LIN {X 0,Y 142.327,Z 764.935,A -85,B 0,C 180,E1 7207.887,E2 7207.887} C_VEL
LIN {X 0,Y 140.279,Z 766.739,A -85,B 0,C 180,E1 7204.976,E2 7204.976} C_VEL
LIN {X 0,Y 137.442,Z 769.448,A -85,B 0,C 180,E1 7201.685,E2 7201.685} C_VEL
LIN {X 0,Y 130.762,Z 776.335,A -85,B 0,C 180,E1 7194.167,E2 7194.167} C_VEL
LIN {X 0,Y 129.959,Z 778.072,A -85,B 0,C 180,E1 7191.372,E2 7191.372} C_VEL
LIN {X 0,Y 136.056,Z 784.68,A -85,B 0,C 180,E1 7176.161,E2 7176.161} C_VEL
LIN {X 0,Y 149.948,Z 789.28,A -85,B 0,C 180,E1 7165.01,E2 7165.01} C_VEL
LIN {X 0,Y 152.41,Z 789.916,A -85,B 0,C 180,E1 7163.584,E2 7163.584} C_VEL
LIN {X 0,Y 141.835,Z 799.917,A -85,B 0,C 180,E1 7157.151,E2 7157.151} C_VEL
LIN {X 0,Y 132.635,Z 808.523,A -85,B 0,C 180,E1 7149.289,E2 7149.289} C_VEL
LIN {X 0,Y 125.571,Z 815.712,A -85,B 0,C 180,E1 7139.786,E2 7139.786} C_VEL
LIN {X 0,Y 121.824,Z 820.643,A -85,B 0,C 180,E1 7130.164,E2 7130.164} C_VEL
LIN {X 0,Y 120.73,Z 823.658,A -85,B 0,C 180,E1 7120.981,E2 7120.981} C_VEL
LIN {X 0,Y 120.991,Z 824.935,A -85,B 0,C 180,E1 7113.791,E2 7113.791} C_VEL
LIN {X 0,Y 121.063,Z 825.276,A -85,B 0,C 180,E1 7108.107,E2 7108.107} C_VEL
LIN {X 0,Y 120.709,Z 824.803,A -85,B 0,C 180,E1 7101.425,E2 7101.425} C_VEL
LIN {X 0,Y 121.285,Z 822.901,A -85,B 0,C 180,E1 7092.24,E2 7092.24} C_VEL
LIN {X 0,Y 124.517,Z 819.128,A -85,B 0,C 180,E1 7082.242,E2 7082.242} C_VEL
LIN {X 0,Y 130.8,Z 813.597,A -85,B 0,C 180,E1 7072.85,E2 7072.85} C_VEL
LIN {X 0,Y 139.988,Z 806.145,A -85,B 0,C 180,E1 7064.418,E2 7064.418} C_VEL
LIN {X 0,Y 151.07,Z 797.105,A -85,B 0,C 180,E1 7057.417,E2 7057.417} C_VEL
LIN {X 0,Y 163.41,Z 786.509,A -85,B 0,C 180,E1 7051.635,E2 7051.635} C_VEL
LIN {X 0,Y 148.498,Z 786.74,A -85,B 0,C 180,E1 7044.634,E2 7044.634} C_VEL
LIN {X 0,Y 138.257,Z 785.962,A -85,B 0,C 180,E1 7036.381,E2 7036.381} C_VEL
LIN {X 0,Y 132.254,Z 784.513,A -85,B 0,C 180,E1 7026.51,E2 7026.51} C_VEL
LIN {X 0,Y 131.134,Z 783.114,A -85,B 0,C 180,E1 7018.688,E2 7018.688} C_VEL
LIN {X 0,Y 134.316,Z 780.824,A -85,B 0,C 180,E1 7007.531,E2 7007.531} C_VEL
LIN {X 0,Y 143.154,Z 778.008,A -85,B 0,C 180,E1 6997.408,E2 6997.408} C_VEL
LIN {X 0,Y 155.053,Z 775.028,A -85,B 0,C 180,E1 6989.801,E2 6989.801} C_VEL
LIN {X 0,Y 165.287,Z 772.555,A -85,B 0,C 180,E1 6985.356,E2 6985.356} C_VEL
LIN {X 0,Y 153.328,Z 781.917,A -85,B 0,C 180,E1 6979.727,E2 6979.727} C_VEL
LIN {X 0,Y 142.444,Z 789.724,A -85,B 0,C 180,E1 6972.913,E2 6972.913} C_VEL
LIN {X 0,Y 133.258,Z 795.917,A -85,B 0,C 180,E1 6964.768,E2 6964.768} C_VEL
LIN {X 0,Y 126.676,Z 800.222,A -85,B 0,C 180,E1 6955.73,E2 6955.73} C_VEL
LIN {X 0,Y 122.964,Z 802.645,A -85,B 0,C 180,E1 6946.535,E2 6946.535} C_VEL
LIN {X 0,Y 121.464,Z 803.514,A -85,B 0,C 180,E1 6937.569,E2 6937.569} C_VEL
LIN {X 0,Y 121.376,Z 803.12,A -85,B 0,C 180,E1 6929.056,E2 6929.056} C_VEL
LIN {X 0,Y 122.613,Z 801.434,A -85,B 0,C 180,E1 6920.14,E2 6920.14} C_VEL
LIN {X 0,Y 125.928,Z 798.163,A -85,B 0,C 180,E1 6911.002,E2 6911.002} C_VEL
LIN {X 0,Y 131.607,Z 793.272,A -85,B 0,C 180,E1 6902.391,E2 6902.391} C_VEL
LIN {X 0,Y 140.034,Z 786.271,A -85,B 0,C 180,E1 6894.162,E2 6894.162} C_VEL
LIN {X 0,Y 149.617,Z 778.131,A -85,B 0,C 180,E1 6887.549,E2 6887.549} C_VEL
LIN {X 0,Y 160.16,Z 768.649,A -85,B 0,C 180,E1 6882.02,E2 6882.02} C_VEL
LIN {X 0,Y 171.365,Z 757.748,A -85,B 0,C 180,E1 6877.361,E2 6877.361} C_VEL
LIN {X 0,Y 183.117,Z 745.114,A -85,B 0,C 180,E1 6873.301,E2 6873.301} C_VEL
LIN {X 0,Y 172.911,Z 750.159,A -85,B 0,C 180,E1 6870.589,E2 6870.589} C_VEL
LIN {X 0,Y 159.994,Z 756.362,A -85,B 0,C 180,E1 6865.854,E2 6865.854} C_VEL
LIN {X 0,Y 149.86,Z 761.284,A -85,B 0,C 180,E1 6860.71,E2 6860.71} C_VEL
LIN {X 0,Y 142.024,Z 765.507,A -85,B 0,C 180,E1 6855.1,E2 6855.1} C_VEL
LIN {X 0,Y 136.055,Z 769.276,A -85,B 0,C 180,E1 6848.879,E2 6848.879} C_VEL
LIN {X 0,Y 132.224,Z 772.647,A -85,B 0,C 180,E1 6842.602,E2 6842.602} C_VEL
LIN {X 0,Y 130.123,Z 776.685,A -85,B 0,C 180,E1 6834.269,E2 6834.269} C_VEL
LIN {X 0,Y 129.959,Z 778.072,A -85,B 0,C 180,E1 6831.372,E2 6831.372} C_VEL
LIN {X 0,Y 129.127,Z 780.467,A -85,B 0,C 180,E1 6827.59,E2 6827.59} C_VEL
LIN {X 0,Y 127.185,Z 786.25,A -85,B 0,C 180,E1 6819.802,E2 6819.802} C_VEL
LIN {X 0,Y 128.371,Z 787.985,A -85,B 0,C 180,E1 6816.472,E2 6816.472} C_VEL
LIN {X 0,Y 128.538,Z 788.078,A -85,B 0,C 180,E1 6816.241,E2 6816.241} C_VEL
LIN {X 0,Y 141.942,Z 792.523,A -85,B 0,C 180,E1 6804.718,E2 6804.718} C_VEL
LIN {X 0,Y 143.15,Z 792.902,A -85,B 0,C 180,E1 6803.903,E2 6803.903} C_VEL
LIN {X 0,Y 131.986,Z 802.686,A -85,B 0,C 180,E1 6796.657,E2 6796.657} C_VEL
LIN {X 0,Y 122.988,Z 810.577,A -85,B 0,C 180,E1 6788.16,E2 6788.16} C_VEL
LIN {X 0,Y 116.513,Z 816.869,A -85,B 0,C 180,E1 6778.163,E2 6778.163} C_VEL
LIN {X 0,Y 113.291,Z 821.249,A -85,B 0,C 180,E1 6767.611,E2 6767.611} C_VEL
LIN {X 0,Y 112.786,Z 823.617,A -85,B 0,C 180,E1 6758.154,E2 6758.154} C_VEL
LIN {X 0,Y 113.119,Z 824.457,A -85,B 0,C 180,E1 6751.519,E2 6751.519} C_VEL
LIN {X 0,Y 112.949,Z 824.477,A -85,B 0,C 180,E1 6745.43,E2 6745.43} C_VEL
LIN {X 0,Y 112.786,Z 823.47,A -85,B 0,C 180,E1 6736.674,E2 6736.674} C_VEL
LIN {X 0,Y 114.786,Z 820.705,A -85,B 0,C 180,E1 6726.147,E2 6726.147} C_VEL
LIN {X 0,Y 120.346,Z 815.871,A -85,B 0,C 180,E1 6715.334,E2 6715.334} C_VEL
LIN {X 0,Y 129.16,Z 809.22,A -85,B 0,C 180,E1 6705.835,E2 6705.835} C_VEL
LIN {X 0,Y 140.544,Z 800.671,A -85,B 0,C 180,E1 6697.844,E2 6697.844} C_VEL
LIN {X 0,Y 153.385,Z 790.579,A -85,B 0,C 180,E1 6691.431,E2 6691.431} C_VEL
LIN {X 0,Y 139.962,Z 790.459,A -85,B 0,C 180,E1 6684.476,E2 6684.476} C_VEL
LIN {X 0,Y 130.135,Z 789.445,A -85,B 0,C 180,E1 6675.598,E2 6675.598} C_VEL
LIN {X 0,Y 125.2,Z 788.207,A -85,B 0,C 180,E1 6666.878,E2 6666.878} C_VEL
LIN {X 0,Y 124.752,Z 785.827,A -85,B 0,C 180,E1 6653.093,E2 6653.093} C_VEL
LIN {X 0,Y 134.755,Z 782.281,A -85,B 0,C 180,E1 6637.763,E2 6637.763} C_VEL
LIN {X 0,Y 148.914,Z 778.871,A -85,B 0,C 180,E1 6628.416,E2 6628.416} C_VEL
LIN {X 0,Y 155.328,Z 777.427,A -85,B 0,C 180,E1 6625.483,E2 6625.483} C_VEL
LIN {X 0,Y 142.741,Z 786.385,A -85,B 0,C 180,E1 6619.158,E2 6619.158} C_VEL
LIN {X 0,Y 132.024,Z 793.328,A -85,B 0,C 180,E1 6611.794,E2 6611.794} C_VEL
LIN {X 0,Y 123.207,Z 798.686,A -85,B 0,C 180,E1 6602.938,E2 6602.938} C_VEL
LIN {X 0,Y 117.214,Z 802.205,A -85,B 0,C 180,E1 6593.104,E2 6593.104} C_VEL
LIN {X 0,Y 114.199,Z 803.931,A -85,B 0,C 180,E1 6583.159,E2 6583.159} C_VEL
LIN {X 0,Y 113.323,Z 804.205,A -85,B 0,C 180,E1 6574.048,E2 6574.048} C_VEL
LIN {X 0,Y 113.769,Z 803.328,A -85,B 0,C 180,E1 6564.958,E2 6564.958} C_VEL
LIN {X 0,Y 115.926,Z 801.107,A -85,B 0,C 180,E1 6555.515,E2 6555.515} C_VEL
LIN {X 0,Y 120.867,Z 796.979,A -85,B 0,C 180,E1 6545.567,E2 6545.567} C_VEL
LIN {X 0,Y 128.146,Z 791.351,A -85,B 0,C 180,E1 6536.895,E2 6536.895} C_VEL
LIN {X 0,Y 137.71,Z 783.926,A -85,B 0,C 180,E1 6529.197,E2 6529.197} C_VEL
LIN {X 0,Y 148.674,Z 774.977,A -85,B 0,C 180,E1 6522.787,E2 6522.787} C_VEL
LIN {X 0,Y 160.252,Z 764.773,A -85,B 0,C 180,E1 6517.59,E2 6517.59} C_VEL
LIN {X 0,Y 172.115,Z 753.272,A -85,B 0,C 180,E1 6513.296,E2 6513.296} C_VEL
LIN {X 0,Y 156.016,Z 760.477,A -85,B 0,C 180,E1 6507.895,E2 6507.895} C_VEL
LIN {X 0,Y 144.573,Z 765.541,A -85,B 0,C 180,E1 6502.359,E2 6502.359} C_VEL
LIN {X 0,Y 136.263,Z 769.637,A -85,B 0,C 180,E1 6496.63,E2 6496.63} C_VEL
LIN {X 0,Y 129.858,Z 773.325,A -85,B 0,C 180,E1 6490.202,E2 6490.202} C_VEL
LIN {X 0,Y 125.481,Z 776.754,A -85,B 0,C 180,E1 6483.199,E2 6483.199} C_VEL
LIN {X 0,Y 123.17,Z 780.474,A -85,B 0,C 180,E1 6474.879,E2 6474.879} C_VEL
LIN {X 0,Y 124.08,Z 784.569,A -85,B 0,C 180,E1 6465.059,E2 6465.059} C_VEL
LIN {X 0,Y 128.538,Z 788.078,A -85,B 0,C 180,E1 6456.241,E2 6456.241} C_VEL
LIN {X 0,Y 129.404,Z 789.371,A -85,B 0,C 180,E1 6454.005,E2 6454.005} C_VEL
LIN {X 0,Y 129.566,Z 793.797,A -85,B 0,C 180,E1 6448.256,E2 6448.256} C_VEL
LIN {X 0,Y 131.281,Z 794.906,A -85,B 0,C 180,E1 6446.152,E2 6446.152} C_VEL
LIN {X 0,Y 133.864,Z 795.665,A -85,B 0,C 180,E1 6444.259,E2 6444.259} C_VEL
LIN {X 0,Y 122.64,Z 804.754,A -85,B 0,C 180,E1 6436.519,E2 6436.519} C_VEL
LIN {X 0,Y 113.746,Z 812.064,A -85,B 0,C 180,E1 6427.339,E2 6427.339} C_VEL
LIN {X 0,Y 107.834,Z 817.537,A -85,B 0,C 180,E1 6417.022,E2 6417.022} C_VEL
LIN {X 0,Y 105.071,Z 821.303,A -85,B 0,C 180,E1 6406.019,E2 6406.019} C_VEL
LIN {X 0,Y 104.914,Z 823.292,A -85,B 0,C 180,E1 6396.017,E2 6396.017} C_VEL
LIN {X 0,Y 105.176,Z 823.802,A -85,B 0,C 180,E1 6389.455,E2 6389.455} C_VEL
LIN {X 0,Y 104.791,Z 823.598,A -85,B 0,C 180,E1 6382.323,E2 6382.323} C_VEL
LIN {X 0,Y 105.338,Z 821.994,A -85,B 0,C 180,E1 6371.745,E2 6371.745} C_VEL
LIN {X 0,Y 109.014,Z 818.561,A -85,B 0,C 180,E1 6360.311,E2 6360.311} C_VEL
LIN {X 0,Y 116.195,Z 813.317,A -85,B 0,C 180,E1 6349.805,E2 6349.805} C_VEL
LIN {X 0,Y 126.551,Z 806.237,A -85,B 0,C 180,E1 6340.669,E2 6340.669} C_VEL
LIN {X 0,Y 138.833,Z 797.607,A -85,B 0,C 180,E1 6333.339,E2 6333.339} C_VEL
LIN {X 0,Y 143.313,Z 794.292,A -85,B 0,C 180,E1 6331.198,E2 6331.198} C_VEL
LIN {X 0,Y 129.824,Z 793.788,A -85,B 0,C 180,E1 6323.126,E2 6323.126} C_VEL
LIN {X 0,Y 118.498,Z 791.93,A -85,B 0,C 180,E1 6308.734,E2 6308.734} C_VEL
LIN {X 0,Y 117.735,Z 789.183,A -85,B 0,C 180,E1 6292.189,E2 6292.189} C_VEL
LIN {X 0,Y 128.54,Z 785.675,A -85,B 0,C 180,E1 6276.139,E2 6276.139} C_VEL
LIN {X 0,Y 144.073,Z 782.191,A -85,B 0,C 180,E1 6266.274,E2 6266.274} C_VEL
LIN {X 0,Y 145.349,Z 781.942,A -85,B 0,C 180,E1 6265.638,E2 6265.638} C_VEL
LIN {X 0,Y 132.716,Z 790.085,A -85,B 0,C 180,E1 6258.885,E2 6258.885} C_VEL
LIN {X 0,Y 121.618,Z 796.572,A -85,B 0,C 180,E1 6250.503,E2 6250.503} C_VEL
LIN {X 0,Y 113.234,Z 801.123,A -85,B 0,C 180,E1 6240.807,E2 6240.807} C_VEL
LIN {X 0,Y 107.93,Z 803.88,A -85,B 0,C 180,E1 6230.046,E2 6230.046} C_VEL
LIN {X 0,Y 105.668,Z 804.929,A -85,B 0,C 180,E1 6219.257,E2 6219.257} C_VEL
LIN {X 0,Y 105.392,Z 804.699,A -85,B 0,C 180,E1 6210,E2 6210} C_VEL
LIN {X 0,Y 106.563,Z 803.319,A -85,B 0,C 180,E1 6200.277,E2 6200.277} C_VEL
LIN {X 0,Y 110.166,Z 800.347,A -85,B 0,C 180,E1 6189.825,E2 6189.825} C_VEL
LIN {X 0,Y 116.875,Z 795.483,A -85,B 0,C 180,E1 6179.686,E2 6179.686} C_VEL
LIN {X 0,Y 125.861,Z 789.097,A -85,B 0,C 180,E1 6171.128,E2 6171.128} C_VEL
LIN {X 0,Y 136.419,Z 781.311,A -85,B 0,C 180,E1 6164.088,E2 6164.088} C_VEL
LIN {X 0,Y 148.581,Z 771.642,A -85,B 0,C 180,E1 6158.062,E2 6158.062} C_VEL
LIN {X 0,Y 161.347,Z 760.482,A -85,B 0,C 180,E1 6153.142,E2 6153.142} C_VEL
LIN {X 0,Y 151.263,Z 764.693,A -85,B 0,C 180,E1 6149.721,E2 6149.721} C_VEL
LIN {X 0,Y 139.888,Z 769.384,A -85,B 0,C 180,E1 6144.493,E2 6144.493} C_VEL
LIN {X 0,Y 130.482,Z 773.549,A -85,B 0,C 180,E1 6138.313,E2 6138.313} C_VEL
LIN {X 0,Y 123.628,Z 777.186,A -85,B 0,C 180,E1 6131.667,E2 6131.667} C_VEL
LIN {X 0,Y 118.817,Z 780.496,A -85,B 0,C 180,E1 6124.345,E2 6124.345} C_VEL
LIN {X 0,Y 116.124,Z 784.251,A -85,B 0,C 180,E1 6115.062,E2 6115.062} C_VEL
LIN {X 0,Y 117.022,Z 788.236,A -85,B 0,C 180,E1 6104.643,E2 6104.643} C_VEL
LIN {X 0,Y 124.71,Z 792.903,A -85,B 0,C 180,E1 6091.771,E2 6091.771} C_VEL
LIN {X 0,Y 131.281,Z 794.906,A -85,B 0,C 180,E1 6086.152,E2 6086.152} C_VEL
LIN {X 0,Y 131.585,Z 795.64,A -85,B 0,C 180,E1 6085.153,E2 6085.153} C_VEL
LIN {X 0,Y 130.245,Z 797.057,A -85,B 0,C 180,E1 6083.974,E2 6083.974} C_VEL
LIN {X 0,Y 126.747,Z 799.167,A -85,B 0,C 180,E1 6082.605,E2 6082.605} C_VEL
LIN {X 0,Y 118.25,Z 803.234,A -85,B 0,C 180,E1 6080.011,E2 6080.011} C_VEL
LIN {X 0,Y 116.114,Z 804.555,A -85,B 0,C 180,E1 6078.768,E2 6078.768} C_VEL
LIN {X 0,Y 106.417,Z 811.832,A -85,B 0,C 180,E1 6069.014,E2 6069.014} C_VEL
LIN {X 0,Y 99.818,Z 817.385,A -85,B 0,C 180,E1 6057.437,E2 6057.437} C_VEL
LIN {X 0,Y 97.024,Z 820.956,A -85,B 0,C 180,E1 6045.541,E2 6045.541} C_VEL
LIN {X 0,Y 96.982,Z 822.68,A -85,B 0,C 180,E1 6035.324,E2 6035.324} C_VEL
LIN {X 0,Y 97.205,Z 823.082,A -85,B 0,C 180,E1 6029.41,E2 6029.41} C_VEL
LIN {X 0,Y 96.815,Z 822.91,A -85,B 0,C 180,E1 6022.284,E2 6022.284} C_VEL
LIN {X 0,Y 97.474,Z 821.379,A -85,B 0,C 180,E1 6010.837,E2 6010.837} C_VEL
LIN {X 0,Y 101.605,Z 818.045,A -85,B 0,C 180,E1 5998.563,E2 5998.563} C_VEL
LIN {X 0,Y 109.495,Z 812.893,A -85,B 0,C 180,E1 5987.488,E2 5987.488} C_VEL
LIN {X 0,Y 120.665,Z 805.879,A -85,B 0,C 180,E1 5978.075,E2 5978.075} C_VEL
LIN {X 0,Y 133.116,Z 797.639,A -85,B 0,C 180,E1 5970.855,E2 5970.855} C_VEL
LIN {X 0,Y 119.37,Z 796.719,A -85,B 0,C 180,E1 5961.109,E2 5961.109} C_VEL
LIN {X 0,Y 110.948,Z 795.031,A -85,B 0,C 180,E1 5948.289,E2 5948.289} C_VEL
LIN {X 0,Y 110.474,Z 792.426,A -85,B 0,C 180,E1 5931.672,E2 5931.672} C_VEL
LIN {X 0,Y 121.869,Z 788.946,A -85,B 0,C 180,E1 5914.744,E2 5914.744} C_VEL
LIN {X 0,Y 135.348,Z 786.121,A -85,B 0,C 180,E1 5905.832,E2 5905.832} C_VEL
LIN {X 0,Y 122.667,Z 793.471,A -85,B 0,C 180,E1 5898.582,E2 5898.582} C_VEL
LIN {X 0,Y 111.691,Z 799.236,A -85,B 0,C 180,E1 5889.465,E2 5889.465} C_VEL
LIN {X 0,Y 103.665,Z 803.11,A -85,B 0,C 180,E1 5878.833,E2 5878.833} C_VEL
LIN {X 0,Y 99.147,Z 805.155,A -85,B 0,C 180,E1 5867.611,E2 5867.611} C_VEL
LIN {X 0,Y 97.511,Z 805.715,A -85,B 0,C 180,E1 5857.068,E2 5857.068} C_VEL
LIN {X 0,Y 97.599,Z 805.136,A -85,B 0,C 180,E1 5847.064,E2 5847.064} C_VEL
LIN {X 0,Y 99.603,Z 803.296,A -85,B 0,C 180,E1 5836.059,E2 5836.059} C_VEL
LIN {X 0,Y 104.469,Z 799.877,A -85,B 0,C 180,E1 5825.095,E2 5825.095} C_VEL
LIN {X 0,Y 112.23,Z 794.841,A -85,B 0,C 180,E1 5815.237,E2 5815.237} C_VEL
LIN {X 0,Y 122.526,Z 788.079,A -85,B 0,C 180,E1 5806.727,E2 5806.727} C_VEL
LIN {X 0,Y 134.885,Z 779.433,A -85,B 0,C 180,E1 5799.563,E2 5799.563} C_VEL
LIN {X 0,Y 148.116,Z 769.16,A -85,B 0,C 180,E1 5793.868,E2 5793.868} C_VEL
LIN {X 0,Y 150.282,Z 767.348,A -85,B 0,C 180,E1 5793.065,E2 5793.065} C_VEL
LIN {X 0,Y 134.711,Z 773.297,A -85,B 0,C 180,E1 5786.447,E2 5786.447} C_VEL
LIN {X 0,Y 124.392,Z 777.425,A -85,B 0,C 180,E1 5779.873,E2 5779.873} C_VEL
LIN {X 0,Y 117.351,Z 780.792,A -85,B 0,C 180,E1 5773.302,E2 5773.302} C_VEL
LIN {X 0,Y 111.904,Z 784.218,A -85,B 0,C 180,E1 5765.128,E2 5765.128} C_VEL
LIN {X 0,Y 108.991,Z 787.657,A -85,B 0,C 180,E1 5755.793,E2 5755.793} C_VEL
LIN {X 0,Y 109.85,Z 791.651,A -85,B 0,C 180,E1 5744.155,E2 5744.155} C_VEL
LIN {X 0,Y 117.483,Z 796.065,A -85,B 0,C 180,E1 5730.983,E2 5730.983} C_VEL
LIN {X 0,Y 124.676,Z 798.141,A -85,B 0,C 180,E1 5724.733,E2 5724.733} C_VEL
LIN {X 0,Y 116.114,Z 804.555,A -85,B 0,C 180,E1 5718.768,E2 5718.768} C_VEL
LIN {X 0,Y 111.632,Z 807.293,A -85,B 0,C 180,E1 5715.891,E2 5715.891} C_VEL
LIN {X 0,Y 97.65,Z 813.239,A -85,B 0,C 180,E1 5707.704,E2 5707.704} C_VEL
LIN {X 0,Y 94.735,Z 814.833,A -85,B 0,C 180,E1 5704.259,E2 5704.259} C_VEL
LIN {X 0,Y 89.936,Z 819.134,A -85,B 0,C 180,E1 5691.523,E2 5691.523} C_VEL
LIN {X 0,Y 88.829,Z 821.577,A -85,B 0,C 180,E1 5679.066,E2 5679.066} C_VEL
LIN {X 0,Y 89.213,Z 822.314,A -85,B 0,C 180,E1 5671.284,E2 5671.284} C_VEL
LIN {X 0,Y 88.99,Z 822.354,A -85,B 0,C 180,E1 5664.843,E2 5664.843} C_VEL
LIN {X 0,Y 89.061,Z 821.415,A -85,B 0,C 180,E1 5653.7,E2 5653.7} C_VEL
LIN {X 0,Y 92.282,Z 818.805,A -85,B 0,C 180,E1 5640.819,E2 5640.819} C_VEL
LIN {X 0,Y 99.688,Z 814.332,A -85,B 0,C 180,E1 5628.549,E2 5628.549} C_VEL
LIN {X 0,Y 111.313,Z 807.695,A -85,B 0,C 180,E1 5617.771,E2 5617.771} C_VEL
LIN {X 0,Y 123.104,Z 800.647,A -85,B 0,C 180,E1 5610.526,E2 5610.526} C_VEL
LIN {X 0,Y 110.365,Z 799.48,A -85,B 0,C 180,E1 5600.135,E2 5600.135} C_VEL
LIN {X 0,Y 103.467,Z 797.974,A -85,B 0,C 180,E1 5588.333,E2 5588.333} C_VEL
LIN {X 0,Y 103.134,Z 795.448,A -85,B 0,C 180,E1 5571.074,E2 5571.074} C_VEL
LIN {X 0,Y 115.694,Z 791.888,A -85,B 0,C 180,E1 5552.737,E2 5552.737} C_VEL
LIN {X 0,Y 125.218,Z 790.042,A -85,B 0,C 180,E1 5546.015,E2 5546.015} C_VEL
LIN {X 0,Y 112.006,Z 796.859,A -85,B 0,C 180,E1 5537.811,E2 5537.811} C_VEL
LIN {X 0,Y 101.314,Z 801.806,A -85,B 0,C 180,E1 5527.726,E2 5527.726} C_VEL
LIN {X 0,Y 93.907,Z 804.94,A -85,B 0,C 180,E1 5515.884,E2 5515.884} C_VEL
LIN {X 0,Y 90.253,Z 806.307,A -85,B 0,C 180,E1 5503.453,E2 5503.453} C_VEL
LIN {X 0,Y 89.401,Z 806.281,A -85,B 0,C 180,E1 5492.564,E2 5492.564} C_VEL
LIN {X 0,Y 90.262,Z 805.262,A -85,B 0,C 180,E1 5481.721,E2 5481.721} C_VEL
LIN {X 0,Y 93.906,Z 802.719,A -85,B 0,C 180,E1 5469.429,E2 5469.429} C_VEL
LIN {X 0,Y 101.16,Z 798.371,A -85,B 0,C 180,E1 5457.742,E2 5457.742} C_VEL
LIN {X 0,Y 111.001,Z 792.525,A -85,B 0,C 180,E1 5448.197,E2 5448.197} C_VEL
LIN {X 0,Y 123.162,Z 784.885,A -85,B 0,C 180,E1 5440.26,E2 5440.26} C_VEL
LIN {X 0,Y 136.367,Z 775.768,A -85,B 0,C 180,E1 5434.052,E2 5434.052} C_VEL
LIN {X 0,Y 139.253,Z 773.525,A -85,B 0,C 180,E1 5432.806,E2 5432.806} C_VEL
LIN {X 0,Y 128.944,Z 777.191,A -85,B 0,C 180,E1 5428.232,E2 5428.232} C_VEL
LIN {X 0,Y 119.028,Z 780.834,A -85,B 0,C 180,E1 5422.212,E2 5422.212} C_VEL
LIN {X 0,Y 110.702,Z 784.375,A -85,B 0,C 180,E1 5414.651,E2 5414.651} C_VEL
LIN {X 0,Y 105.118,Z 787.545,A -85,B 0,C 180,E1 5406.556,E2 5406.556} C_VEL
LIN {X 0,Y 101.745,Z 791.023,A -85,B 0,C 180,E1 5396.058,E2 5396.058} C_VEL
LIN {X 0,Y 102.408,Z 794.702,A -85,B 0,C 180,E1 5384.137,E2 5384.137} C_VEL
LIN {X 0,Y 111.081,Z 799.293,A -85,B 0,C 180,E1 5369.134,E2 5369.134} C_VEL
LIN {X 0,Y 115.287,Z 800.561,A -85,B 0,C 180,E1 5365.158,E2 5365.158} C_VEL
LIN {X 0,Y 103.854,Z 808.358,A -85,B 0,C 180,E1 5356.12,E2 5356.12} C_VEL
LIN {X 0,Y 94.957,Z 814.662,A -85,B 0,C 180,E1 5344.653,E2 5344.653} C_VEL
LIN {X 0,Y 94.735,Z 814.833,A -85,B 0,C 180,E1 5344.259,E2 5344.259} C_VEL
LIN {X 0,Y 91.625,Z 816.539,A -85,B 0,C 180,E1 5340.012,E2 5340.012} C_VEL
LIN {X 0,Y 84.273,Z 818.948,A -85,B 0,C 180,E1 5331.523,E2 5331.523} C_VEL
LIN {X 0,Y 81.129,Z 820.124,A -85,B 0,C 180,E1 5324.927,E2 5324.927} C_VEL
LIN {X 0,Y 80.882,Z 820.397,A -85,B 0,C 180,E1 5322.967,E2 5322.967} C_VEL
LIN {X 0,Y 81.168,Z 821.517,A -85,B 0,C 180,E1 5312.824,E2 5312.824} C_VEL
LIN {X 0,Y 81.157,Z 821.671,A -85,B 0,C 180,E1 5307.175,E2 5307.175} C_VEL
LIN {X 0,Y 80.91,Z 821.063,A -85,B 0,C 180,E1 5295.69,E2 5295.69} C_VEL
LIN {X 0,Y 83.789,Z 818.853,A -85,B 0,C 180,E1 5281.489,E2 5281.489} C_VEL
LIN {X 0,Y 91.227,Z 814.826,A -85,B 0,C 180,E1 5268.043,E2 5268.043} C_VEL
LIN {X 0,Y 102.576,Z 809.014,A -85,B 0,C 180,E1 5256.937,E2 5256.937} C_VEL
LIN {X 0,Y 112.986,Z 803.32,A -85,B 0,C 180,E1 5250.053,E2 5250.053} C_VEL
LIN {X 0,Y 98.12,Z 801.427,A -85,B 0,C 180,E1 5234.154,E2 5234.154} C_VEL
LIN {X 0,Y 94.598,Z 799.248,A -85,B 0,C 180,E1 5217.575,E2 5217.575} C_VEL
LIN {X 0,Y 100.27,Z 796.673,A -85,B 0,C 180,E1 5200.786,E2 5200.786} C_VEL
LIN {X 0,Y 115.285,Z 793.547,A -85,B 0,C 180,E1 5186.368,E2 5186.368} C_VEL
LIN {X 0,Y 101.905,Z 799.653,A -85,B 0,C 180,E1 5177.382,E2 5177.382} C_VEL
LIN {X 0,Y 91.4,Z 803.887,A -85,B 0,C 180,E1 5166.209,E2 5166.209} C_VEL
LIN {X 0,Y 84.56,Z 806.349,A -85,B 0,C 180,E1 5152.968,E2 5152.968} C_VEL
LIN {X 0,Y 81.781,Z 807.116,A -85,B 0,C 180,E1 5139.856,E2 5139.856} C_VEL
LIN {X 0,Y 81.588,Z 806.709,A -85,B 0,C 180,E1 5127.893,E2 5127.893} C_VEL
LIN {X 0,Y 83.604,Z 805.194,A -85,B 0,C 180,E1 5115.455,E2 5115.455} C_VEL
LIN {X 0,Y 89.096,Z 802.065,A -85,B 0,C 180,E1 5102.606,E2 5102.606} C_VEL
LIN {X 0,Y 97.926,Z 797.337,A -85,B 0,C 180,E1 5091.477,E2 5091.477} C_VEL
LIN {X 0,Y 110.125,Z 790.535,A -85,B 0,C 180,E1 5081.883,E2 5081.883} C_VEL
LIN {X 0,Y 123.847,Z 782.156,A -85,B 0,C 180,E1 5074.565,E2 5074.565} C_VEL
LIN {X 0,Y 128.184,Z 779.257,A -85,B 0,C 180,E1 5072.637,E2 5072.637} C_VEL
LIN {X 0,Y 113.405,Z 784.188,A -85,B 0,C 180,E1 5064.483,E2 5064.483} C_VEL
LIN {X 0,Y 104.295,Z 787.633,A -85,B 0,C 180,E1 5056.526,E2 5056.526} C_VEL
LIN {X 0,Y 98.041,Z 790.777,A -85,B 0,C 180,E1 5047.621,E2 5047.621} C_VEL
LIN {X 0,Y 94.456,Z 794.024,A -85,B 0,C 180,E1 5036.968,E2 5036.968} C_VEL
LIN {X 0,Y 95.069,Z 797.698,A -85,B 0,C 180,E1 5023.505,E2 5023.505} C_VEL
LIN {X 0,Y 103.869,Z 802.001,A -85,B 0,C 180,E1 5007.898,E2 5007.898} C_VEL
LIN {X 0,Y 105.931,Z 802.689,A -85,B 0,C 180,E1 5005.68,E2 5005.68} C_VEL
LIN {X 0,Y 94.058,Z 810.122,A -85,B 0,C 180,E1 4995.448,E2 4995.448} C_VEL
LIN {X 0,Y 85.508,Z 815.736,A -85,B 0,C 180,E1 4982.662,E2 4982.662} C_VEL
LIN {X 0,Y 81.378,Z 819.418,A -85,B 0,C 180,E1 4968.63,E2 4968.63} C_VEL
LIN {X 0,Y 80.882,Z 820.397,A -85,B 0,C 180,E1 4962.967,E2 4962.967} C_VEL
LIN {X 0,Y 79.979,Z 820.962,A -85,B 0,C 180,E1 4958.291,E2 4958.291} C_VEL
LIN {X 0,Y 77.39,Z 821.241,A -85,B 0,C 180,E1 4952.047,E2 4952.047} C_VEL
LIN {X 0,Y 72.904,Z 820.718,A -85,B 0,C 180,E1 4938.383,E2 4938.383} C_VEL
LIN {X 0,Y 72.882,Z 820.566,A -85,B 0,C 180,E1 4936.572,E2 4936.572} C_VEL
LIN {X 0,Y 75.796,Z 818.577,A -85,B 0,C 180,E1 4920.785,E2 4920.785} C_VEL
LIN {X 0,Y 83.72,Z 814.783,A -85,B 0,C 180,E1 4906.156,E2 4906.156} C_VEL
LIN {X 0,Y 96.448,Z 808.907,A -85,B 0,C 180,E1 4893.968,E2 4893.968} C_VEL
LIN {X 0,Y 102.951,Z 805.671,A -85,B 0,C 180,E1 4889.528,E2 4889.528} C_VEL
LIN {X 0,Y 89.162,Z 803.541,A -85,B 0,C 180,E1 4871.643,E2 4871.643} C_VEL
LIN {X 0,Y 88.461,Z 800.706,A -85,B 0,C 180,E1 4848.919,E2 4848.919} C_VEL
LIN {X 0,Y 103.066,Z 797.216,A -85,B 0,C 180,E1 4828.406,E2 4828.406} C_VEL
LIN {X 0,Y 105.229,Z 796.833,A -85,B 0,C 180,E1 4826.738,E2 4826.738} C_VEL
LIN {X 0,Y 91.78,Z 802.191,A -85,B 0,C 180,E1 4816.879,E2 4816.879} C_VEL
LIN {X 0,Y 81.508,Z 805.728,A -85,B 0,C 180,E1 4804.353,E2 4804.353} C_VEL
LIN {X 0,Y 75.369,Z 807.536,A -85,B 0,C 180,E1 4789.37,E2 4789.37} C_VEL
LIN {X 0,Y 73.511,Z 807.79,A -85,B 0,C 180,E1 4775.464,E2 4775.464} C_VEL
LIN {X 0,Y 74.167,Z 807.024,A -85,B 0,C 180,E1 4762.253,E2 4762.253} C_VEL
LIN {X 0,Y 78.21,Z 804.759,A -85,B 0,C 180,E1 4747.448,E2 4747.448} C_VEL
LIN {X 0,Y 86.547,Z 800.711,A -85,B 0,C 180,E1 4733.9,E2 4733.9} C_VEL
LIN {X 0,Y 98.37,Z 794.853,A -85,B 0,C 180,E1 4722.96,E2 4722.96} C_VEL
LIN {X 0,Y 112.017,Z 787.456,A -85,B 0,C 180,E1 4714.796,E2 4714.796} C_VEL
LIN {X 0,Y 117.162,Z 784.41,A -85,B 0,C 180,E1 4712.305,E2 4712.305} C_VEL
LIN {X 0,Y 100.165,Z 789.885,A -85,B 0,C 180,E1 4701.063,E2 4701.063} C_VEL
LIN {X 0,Y 87.1,Z 796.784,A -85,B 0,C 180,E1 4678.029,E2 4678.029} C_VEL
LIN {X 0,Y 87.663,Z 800.478,A -85,B 0,C 180,E1 4662.752,E2 4662.752} C_VEL
LIN {X 0,Y 96.693,Z 804.518,A -85,B 0,C 180,E1 4646.414,E2 4646.414} C_VEL
LIN {X 0,Y 84.657,Z 811.405,A -85,B 0,C 180,E1 4635.124,E2 4635.124} C_VEL
LIN {X 0,Y 76.638,Z 816.282,A -85,B 0,C 180,E1 4621.457,E2 4621.457} C_VEL
LIN {X 0,Y 73.066,Z 819.447,A -85,B 0,C 180,E1 4605.884,E2 4605.884} C_VEL
LIN {X 0,Y 73.139,Z 820.743,A -85,B 0,C 180,E1 4593.706,E2 4593.706} C_VEL
LIN {X 0,Y 73.208,Z 820.941,A -85,B 0,C 180,E1 4587.651,E2 4587.651} C_VEL
LIN {X 0,Y 72.882,Z 820.566,A -85,B 0,C 180,E1 4576.572,E2 4576.572} C_VEL
LIN {X 0,Y 72.451,Z 819.941,A -85,B 0,C 180,E1 4570.485,E2 4570.485} C_VEL
LIN {X 0,Y 70.778,Z 817.93,A -85,B 0,C 180,E1 4557.608,E2 4557.608} C_VEL
LIN {X 0,Y 72.248,Z 816.416,A -85,B 0,C 180,E1 4550.168,E2 4550.168} C_VEL
LIN {X 0,Y 73.097,Z 816.013,A -85,B 0,C 180,E1 4548.567,E2 4548.567} C_VEL
LIN {X 0,Y 85.17,Z 811.104,A -85,B 0,C 180,E1 4534.736,E2 4534.736} C_VEL
LIN {X 0,Y 93.005,Z 807.723,A -85,B 0,C 180,E1 4528.93,E2 4528.93} C_VEL
LIN {X 0,Y 81.228,Z 805.699,A -85,B 0,C 180,E1 4511.356,E2 4511.356} C_VEL
LIN {X 0,Y 80.942,Z 802.997,A -85,B 0,C 180,E1 4487.875,E2 4487.875} C_VEL
LIN {X 0,Y 95.146,Z 799.794,A -85,B 0,C 180,E1 4467.215,E2 4467.215} C_VEL
LIN {X 0,Y 81.624,Z 804.484,A -85,B 0,C 180,E1 4456.281,E2 4456.281} C_VEL
LIN {X 0,Y 71.664,Z 807.341,A -85,B 0,C 180,E1 4442.018,E2 4442.018} C_VEL
LIN {X 0,Y 66.546,Z 808.499,A -85,B 0,C 180,E1 4425.692,E2 4425.692} C_VEL
LIN {X 0,Y 65.517,Z 808.383,A -85,B 0,C 180,E1 4410.875,E2 4410.875} C_VEL
LIN {X 0,Y 67.204,Z 807.216,A -85,B 0,C 180,E1 4396.229,E2 4396.229} C_VEL
LIN {X 0,Y 73.127,Z 804.534,A -85,B 0,C 180,E1 4380.513,E2 4380.513} C_VEL
LIN {X 0,Y 83.595,Z 800.051,A -85,B 0,C 180,E1 4367.018,E2 4367.018} C_VEL
LIN {X 0,Y 97.275,Z 793.703,A -85,B 0,C 180,E1 4356.703,E2 4356.703} C_VEL
LIN {X 0,Y 105.982,Z 789.198,A -85,B 0,C 180,E1 4351.997,E2 4351.997} C_VEL
LIN {X 0,Y 91.639,Z 793.536,A -85,B 0,C 180,E1 4341.106,E2 4341.106} C_VEL
LIN {X 0,Y 84.052,Z 796.452,A -85,B 0,C 180,E1 4330.975,E2 4330.975} C_VEL
LIN {X 0,Y 79.591,Z 799.445,A -85,B 0,C 180,E1 4318.563,E2 4318.563} C_VEL
LIN {X 0,Y 80.204,Z 803.047,A -85,B 0,C 180,E1 4301.843,E2 4301.843} C_VEL
LIN {X 0,Y 87.254,Z 806.3,A -85,B 0,C 180,E1 4287.105,E2 4287.105} C_VEL
LIN {X 0,Y 75.265,Z 812.451,A -85,B 0,C 180,E1 4274.755,E2 4274.755} C_VEL
LIN {X 0,Y 67.538,Z 816.799,A -85,B 0,C 180,E1 4259.144,E2 4259.144} C_VEL
LIN {X 0,Y 64.904,Z 819.328,A -85,B 0,C 180,E1 4242.455,E2 4242.455} C_VEL
LIN {X 0,Y 65.307,Z 820.172,A -85,B 0,C 180,E1 4230.877,E2 4230.877} C_VEL
LIN {X 0,Y 64.94,Z 820.193,A -85,B 0,C 180,E1 4222.924,E2 4222.924} C_VEL
LIN {X 0,Y 66.011,Z 819.153,A -85,B 0,C 180,E1 4206.807,E2 4206.807} C_VEL
LIN {X 0,Y 72.483,Z 816.272,A -85,B 0,C 180,E1 4189.583,E2 4189.583} C_VEL
LIN {X 0,Y 73.097,Z 816.013,A -85,B 0,C 180,E1 4188.567,E2 4188.567} C_VEL
LIN {X 0,Y 74.535,Z 815.053,A -85,B 0,C 180,E1 4184.736,E2 4184.736} C_VEL
LIN {X 0,Y 76.604,Z 812.162,A -85,B 0,C 180,E1 4174.079,E2 4174.079} C_VEL
LIN {X 0,Y 78.834,Z 811.083,A -85,B 0,C 180,E1 4171.31,E2 4171.31} C_VEL
LIN {X 0,Y 82.983,Z 809.464,A -85,B 0,C 180,E1 4168.026,E2 4168.026} C_VEL
LIN {X 0,Y 73.452,Z 807.708,A -85,B 0,C 180,E1 4151.779,E2 4151.779} C_VEL
LIN {X 0,Y 73.658,Z 804.965,A -85,B 0,C 180,E1 4125.854,E2 4125.854} C_VEL
LIN {X 0,Y 84.877,Z 802.539,A -85,B 0,C 180,E1 4107.709,E2 4107.709} C_VEL
LIN {X 0,Y 71.433,Z 806.475,A -85,B 0,C 180,E1 4095.55,E2 4095.55} C_VEL
LIN {X 0,Y 61.897,Z 808.721,A -85,B 0,C 180,E1 4078.987,E2 4078.987} C_VEL
LIN {X 0,Y 57.908,Z 809.3,A -85,B 0,C 180,E1 4060.949,E2 4060.949} C_VEL
LIN {X 0,Y 57.856,Z 808.786,A -85,B 0,C 180,E1 4045.043,E2 4045.043} C_VEL
LIN {X 0,Y 61.631,Z 807.069,A -85,B 0,C 180,E1 4027.085,E2 4027.085} C_VEL
LIN {X 0,Y 70.796,Z 803.595,A -85,B 0,C 180,E1 4010.54,E2 4010.54} C_VEL
LIN {X 0,Y 83.497,Z 798.556,A -85,B 0,C 180,E1 3998.516,E2 3998.516} C_VEL
LIN {X 0,Y 94.845,Z 793.489,A -85,B 0,C 180,E1 3991.445,E2 3991.445} C_VEL
LIN {X 0,Y 78.01,Z 798.608,A -85,B 0,C 180,E1 3974.856,E2 3974.856} C_VEL
LIN {X 0,Y 71.9,Z 804.825,A -85,B 0,C 180,E1 3943.855,E2 3943.855} C_VEL
LIN {X 0,Y 78.006,Z 807.799,A -85,B 0,C 180,E1 3928.156,E2 3928.156} C_VEL
LIN {X 0,Y 65.861,Z 813.343,A -85,B 0,C 180,E1 3914.294,E2 3914.294} C_VEL
LIN {X 0,Y 58.361,Z 817.25,A -85,B 0,C 180,E1 3895.36,E2 3895.36} C_VEL
LIN {X 0,Y 56.983,Z 819.125,A -85,B 0,C 180,E1 3877.055,E2 3877.055} C_VEL
LIN {X 0,Y 57.322,Z 819.481,A -85,B 0,C 180,E1 3869,E2 3869} C_VEL
LIN {X 0,Y 57.01,Z 819.206,A -85,B 0,C 180,E1 3854.697,E2 3854.697} C_VEL
LIN {X 0,Y 61.162,Z 817.404,A -85,B 0,C 180,E1 3835.098,E2 3835.098} C_VEL
LIN {X 0,Y 71.405,Z 813.794,A -85,B 0,C 180,E1 3818.357,E2 3818.357} C_VEL
LIN {X 0,Y 78.834,Z 811.083,A -85,B 0,C 180,E1 3811.31,E2 3811.31} C_VEL
LIN {X 0,Y 79.417,Z 810.557,A -85,B 0,C 180,E1 3809.717,E2 3809.717} C_VEL
LIN {X 0,Y 78.414,Z 810.141,A -85,B 0,C 180,E1 3807.5,E2 3807.5} C_VEL
LIN {X 0,Y 75.387,Z 809.933,A -85,B 0,C 180,E1 3804.493,E2 3804.493} C_VEL
LIN {X 0,Y 67.936,Z 809.967,A -85,B 0,C 180,E1 3797.862,E2 3797.862} C_VEL
LIN {X 0,Y 66.426,Z 809.758,A -85,B 0,C 180,E1 3795.024,E2 3795.024} C_VEL
LIN {X 0,Y 66.126,Z 806.799,A -85,B 0,C 180,E1 3764.203,E2 3764.203} C_VEL
LIN {X 0,Y 74.93,Z 804.917,A -85,B 0,C 180,E1 3748.637,E2 3748.637} C_VEL
LIN {X 0,Y 60.656,Z 808.337,A -85,B 0,C 180,E1 3733.816,E2 3733.816} C_VEL
LIN {X 0,Y 52.25,Z 809.816,A -85,B 0,C 180,E1 3714.898,E2 3714.898} C_VEL
LIN {X 0,Y 49.603,Z 809.909,A -85,B 0,C 180,E1 3695.785,E2 3695.785} C_VEL
LIN {X 0,Y 50.757,Z 809.148,A -85,B 0,C 180,E1 3677.486,E2 3677.486} C_VEL
LIN {X 0,Y 56.828,Z 807.052,A -85,B 0,C 180,E1 3658.141,E2 3658.141} C_VEL
LIN {X 0,Y 68.628,Z 803.091,A -85,B 0,C 180,E1 3642.01,E2 3642.01} C_VEL
LIN {X 0,Y 83.651,Z 797.417,A -85,B 0,C 180,E1 3630.962,E2 3630.962} C_VEL
LIN {X 0,Y 64.839,Z 803.717,A -85,B 0,C 180,E1 3602.655,E2 3602.655} C_VEL
LIN {X 0,Y 65.151,Z 807.442,A -85,B 0,C 180,E1 3579.334,E2 3579.334} C_VEL
LIN {X 0,Y 68.75,Z 809.13,A -85,B 0,C 180,E1 3569.466,E2 3569.466} C_VEL
LIN {X 0,Y 55.951,Z 814.265,A -85,B 0,C 180,E1 3552.771,E2 3552.771} C_VEL
LIN {X 0,Y 49.574,Z 817.384,A -85,B 0,C 180,E1 3531.287,E2 3531.287} C_VEL
LIN {X 0,Y 49.268,Z 818.704,A -85,B 0,C 180,E1 3512.326,E2 3512.326} C_VEL
LIN {X 0,Y 49.132,Z 818.771,A -85,B 0,C 180,E1 3505.634,E2 3505.634} C_VEL
LIN {X 0,Y 50.08,Z 818.09,A -85,B 0,C 180,E1 3485.211,E2 3485.211} C_VEL
LIN {X 0,Y 57.985,Z 815.649,A -85,B 0,C 180,E1 3463.595,E2 3463.595} C_VEL
LIN {X 0,Y 71.544,Z 811.454,A -85,B 0,C 180,E1 3448.302,E2 3448.302} C_VEL
LIN {X 0,Y 72.985,Z 810.964,A -85,B 0,C 180,E1 3447.021,E2 3447.021} C_VEL
LIN {X 0,Y 66.426,Z 809.758,A -85,B 0,C 180,E1 3435.024,E2 3435.024} C_VEL
LIN {X 0,Y 63.703,Z 809.344,A -85,B 0,C 180,E1 3428.613,E2 3428.613} C_VEL
LIN {X 0,Y 57.455,Z 808.961,A -85,B 0,C 180,E1 3409.842,E2 3409.842} C_VEL
LIN {X 0,Y 58.378,Z 808.47,A -85,B 0,C 180,E1 3402.799,E2 3402.799} C_VEL
LIN {X 0,Y 64.664,Z 807.13,A -85,B 0,C 180,E1 3389.591,E2 3389.591} C_VEL
LIN {X 0,Y 50.413,Z 809.811,A -85,B 0,C 180,E1 3372.403,E2 3372.403} C_VEL
LIN {X 0,Y 42.833,Z 810.696,A -85,B 0,C 180,E1 3349.076,E2 3349.076} C_VEL
LIN {X 0,Y 41.723,Z 810.413,A -85,B 0,C 180,E1 3327.253,E2 3327.253} C_VEL
LIN {X 0,Y 45.713,Z 809.078,A -85,B 0,C 180,E1 3304.059,E2 3304.059} C_VEL
LIN {X 0,Y 56.671,Z 805.965,A -85,B 0,C 180,E1 3283.666,E2 3283.666} C_VEL
LIN {X 0,Y 71.128,Z 801.393,A -85,B 0,C 180,E1 3270.965,E2 3270.965} C_VEL
LIN {X 0,Y 72.453,Z 800.923,A -85,B 0,C 180,E1 3270.02,E2 3270.02} C_VEL
LIN {X 0,Y 57.041,Z 805.886,A -85,B 0,C 180,E1 3243.018,E2 3243.018} C_VEL
LIN {X 0,Y 57.328,Z 809.161,A -85,B 0,C 180,E1 3218.518,E2 3218.518} C_VEL
LIN {X 0,Y 59.523,Z 810.208,A -85,B 0,C 180,E1 3211.184,E2 3211.184} C_VEL
LIN {X 0,Y 47.002,Z 814.607,A -85,B 0,C 180,E1 3192.901,E2 3192.901} C_VEL
LIN {X 0,Y 41.137,Z 817.283,A -85,B 0,C 180,E1 3166.957,E2 3166.957} C_VEL
LIN {X 0,Y 41.402,Z 818.028,A -85,B 0,C 180,E1 3149.999,E2 3149.999} C_VEL
LIN {X 0,Y 41.338,Z 817.789,A -85,B 0,C 180,E1 3130.206,E2 3130.206} C_VEL
LIN {X 0,Y 48.004,Z 816.063,A -85,B 0,C 180,E1 3104.912,E2 3104.912} C_VEL
LIN {X 0,Y 61.684,Z 812.555,A -85,B 0,C 180,E1 3086.933,E2 3086.933} C_VEL
LIN {X 0,Y 62.968,Z 812.17,A -85,B 0,C 180,E1 3085.685,E2 3085.685} C_VEL
LIN {X 0,Y 56.055,Z 809.576,A -85,B 0,C 180,E1 3055.518,E2 3055.518} C_VEL
LIN {X 0,Y 58.378,Z 808.47,A -85,B 0,C 180,E1 3042.799,E2 3042.799} C_VEL
LIN {X 0,Y 58.581,Z 808.346,A -85,B 0,C 180,E1 3039.409,E2 3039.409} C_VEL
LIN {X 0,Y 57.12,Z 808.573,A -85,B 0,C 180,E1 3035.093,E2 3035.093} C_VEL
LIN {X 0,Y 53.821,Z 809.18,A -85,B 0,C 180,E1 3029.859,E2 3029.859} C_VEL
LIN {X 0,Y 47.493,Z 810.182,A -85,B 0,C 180,E1 3022.123,E2 3022.123} C_VEL
LIN {X 0,Y 38.736,Z 811.189,A -85,B 0,C 180,E1 3006.637,E2 3006.637} C_VEL
LIN {X 0,Y 33.834,Z 811.376,A -85,B 0,C 180,E1 2980.214,E2 2980.214} C_VEL
LIN {X 0,Y 34.858,Z 810.763,A -85,B 0,C 180,E1 2955.04,E2 2955.04} C_VEL
LIN {X 0,Y 43.468,Z 808.715,A -85,B 0,C 180,E1 2928.16,E2 2928.16} C_VEL
LIN {X 0,Y 58.68,Z 804.813,A -85,B 0,C 180,E1 2910.747,E2 2910.747} C_VEL
LIN {X 0,Y 61.056,Z 804.109,A -85,B 0,C 180,E1 2908.893,E2 2908.893} C_VEL
LIN {X 0,Y 48.836,Z 810.352,A -85,B 0,C 180,E1 2860.355,E2 2860.355} C_VEL
LIN {X 0,Y 50.418,Z 811.107,A -85,B 0,C 180,E1 2853.599,E2 2853.599} C_VEL
LIN {X 0,Y 37.097,Z 815.082,A -85,B 0,C 180,E1 2830.306,E2 2830.306} C_VEL
LIN {X 0,Y 32.983,Z 816.973,A -85,B 0,C 180,E1 2800.479,E2 2800.479} C_VEL
LIN {X 0,Y 33.303,Z 817.31,A -85,B 0,C 180,E1 2788.279,E2 2788.279} C_VEL
LIN {X 0,Y 34.791,Z 816.869,A -85,B 0,C 180,E1 2758.848,E2 2758.848} C_VEL
LIN {X 0,Y 45.911,Z 814.66,A -85,B 0,C 180,E1 2731.857,E2 2731.857} C_VEL
LIN {X 0,Y 53.065,Z 813.073,A -85,B 0,C 180,E1 2723.775,E2 2723.775} C_VEL
LIN {X 0,Y 50.462,Z 809.952,A -85,B 0,C 180,E1 2681.513,E2 2681.513} C_VEL
LIN {X 0,Y 54.563,Z 809.058,A -85,B 0,C 180,E1 2671.139,E2 2671.139} C_VEL
LIN {X 0,Y 40.672,Z 811.016,A -85,B 0,C 180,E1 2651.588,E2 2651.588} C_VEL
LIN {X 0,Y 38.736,Z 811.189,A -85,B 0,C 180,E1 2646.637,E2 2646.637} C_VEL
LIN {X 0,Y 35.1,Z 811.509,A -85,B 0,C 180,E1 2636.967,E2 2636.967} C_VEL
LIN {X 0,Y 29.535,Z 811.819,A -85,B 0,C 180,E1 2619.62,E2 2619.62} C_VEL
LIN {X 0,Y 27.272,Z 811.543,A -85,B 0,C 180,E1 2592.274,E2 2592.274} C_VEL
LIN {X 0,Y 28.364,Z 811.253,A -85,B 0,C 180,E1 2584.454,E2 2584.454} C_VEL
LIN {X 0,Y 40.058,Z 809.021,A -85,B 0,C 180,E1 2556.991,E2 2556.991} C_VEL
LIN {X 0,Y 49.768,Z 806.879,A -85,B 0,C 180,E1 2546.88,E2 2546.88} C_VEL
LIN {X 0,Y 41.071,Z 811.725,A -85,B 0,C 180,E1 2498.587,E2 2498.587} C_VEL
LIN {X 0,Y 41.293,Z 811.878,A -85,B 0,C 180,E1 2496.943,E2 2496.943} C_VEL
LIN {X 0,Y 28.094,Z 815.103,A -85,B 0,C 180,E1 2469.837,E2 2469.837} C_VEL
LIN {X 0,Y 25.234,Z 816.55,A -85,B 0,C 180,E1 2432.27,E2 2432.27} C_VEL
LIN {X 0,Y 25.058,Z 816.583,A -85,B 0,C 180,E1 2423.124,E2 2423.124} C_VEL
LIN {X 0,Y 30.109,Z 815.824,A -85,B 0,C 180,E1 2383.063,E2 2383.063} C_VEL
LIN {X 0,Y 43.31,Z 813.691,A -85,B 0,C 180,E1 2360.795,E2 2360.795} C_VEL
LIN {X 0,Y 43.832,Z 810.854,A -85,B 0,C 180,E1 2315.752,E2 2315.752} C_VEL
LIN {X 0,Y 44.643,Z 810.689,A -85,B 0,C 180,E1 2313.623,E2 2313.623} C_VEL
LIN {X 0,Y 30.36,Z 812.083,A -85,B 0,C 180,E1 2288.737,E2 2288.737} C_VEL
LIN {X 0,Y 25.698,Z 812.03,A -85,B 0,C 180,E1 2256.704,E2 2256.704} C_VEL
LIN {X 0,Y 28.364,Z 811.253,A -85,B 0,C 180,E1 2224.454,E2 2224.454} C_VEL
LIN {X 0,Y 29.828,Z 810.911,A -85,B 0,C 180,E1 2214.61,E2 2214.61} C_VEL
LIN {X 0,Y 34.824,Z 809.971,A -85,B 0,C 180,E1 2188.866,E2 2188.866} C_VEL
LIN {X 0,Y 37.63,Z 809.446,A -85,B 0,C 180,E1 2184.982,E2 2184.982} C_VEL
LIN {X 0,Y 38.346,Z 809.318,A -85,B 0,C 180,E1 2184.011,E2 2184.011} C_VEL
LIN {X 0,Y 32.281,Z 812.483,A -85,B 0,C 180,E1 2142.103,E2 2142.103} C_VEL
LIN {X 0,Y 18.636,Z 815.119,A -85,B 0,C 180,E1 2106.168,E2 2106.168} C_VEL
LIN {X 0,Y 17.301,Z 815.851,A -85,B 0,C 180,E1 2069.999,E2 2069.999} C_VEL
LIN {X 0,Y 21.766,Z 815.463,A -85,B 0,C 180,E1 2018.653,E2 2018.653} C_VEL
LIN {X 0,Y 33.626,Z 814.062,A -85,B 0,C 180,E1 1996.095,E2 1996.095} C_VEL
LIN {X 0,Y 34.511,Z 812.118,A -85,B 0,C 180,E1 1957.265,E2 1957.265} C_VEL
LIN {X 0,Y 20.517,Z 812.868,A -85,B 0,C 180,E1 1925.791,E2 1925.791} C_VEL
LIN {X 0,Y 18.037,Z 812.544,A -85,B 0,C 180,E1 1880.428,E2 1880.428} C_VEL
LIN {X 0,Y 27.074,Z 811.204,A -85,B 0,C 180,E1 1839.147,E2 1839.147} C_VEL
LIN {X 0,Y 37.63,Z 809.446,A -85,B 0,C 180,E1 1824.982,E2 1824.982} C_VEL
LIN {X 0,Y 38.325,Z 809.347,A -85,B 0,C 180,E1 1822.476,E2 1822.476} C_VEL
LIN {X 0,Y 37.662,Z 809.561,A -85,B 0,C 180,E1 1818.513,E2 1818.513} C_VEL
LIN {X 0,Y 35.206,Z 810.201,A -85,B 0,C 180,E1 1812.495,E2 1812.495} C_VEL
LIN {X 0,Y 29.832,Z 811.543,A -85,B 0,C 180,E1 1802.713,E2 1802.713} C_VEL
LIN {X 0,Y 25.284,Z 812.519,A -85,B 0,C 180,E1 1794.22,E2 1794.22} C_VEL
LIN {X 0,Y 21.88,Z 813.138,A -85,B 0,C 180,E1 1789.001,E2 1789.001} C_VEL
LIN {X 0,Y 9.143,Z 814.957,A -85,B 0,C 180,E1 1729.149,E2 1729.149} C_VEL
LIN {X 0,Y 9.213,Z 815.12,A -85,B 0,C 180,E1 1709.997,E2 1709.997} C_VEL
LIN {X 0,Y 19.101,Z 814.653,A -85,B 0,C 180,E1 1635.162,E2 1635.162} C_VEL
LIN {X 0,Y 24.352,Z 814.171,A -85,B 0,C 180,E1 1627.681,E2 1627.681} C_VEL
LIN {X 0,Y 24.913,Z 813.296,A -85,B 0,C 180,E1 1604.414,E2 1604.414} C_VEL
LIN {X 0,Y 11.068,Z 813.544,A -85,B 0,C 180,E1 1562.825,E2 1562.825} C_VEL
LIN {X 0,Y 12.646,Z 813.003,A -85,B 0,C 180,E1 1490.765,E2 1490.765} C_VEL
LIN {X 0,Y 27.35,Z 811.35,A -85,B 0,C 180,E1 1458.411,E2 1458.411} C_VEL
LIN {X 0,Y 23.904,Z 812.802,A -85,B 0,C 180,E1 1431.354,E2 1431.354} C_VEL
LIN {X 0,Y 21.88,Z 813.138,A -85,B 0,C 180,E1 1429.001,E2 1429.001} C_VEL
LIN {X 0,Y 16.306,Z 813.837,A -85,B 0,C 180,E1 1423.225,E2 1423.225} C_VEL
LIN {X 0,Y 8.129,Z 814.294,A -85,B 0,C 180,E1 1416.422,E2 1416.422} C_VEL
LIN {X 0,Y 2.332,Z 814.384,A -85,B 0,C 180,E1 1276.768,E2 1276.768} C_VEL
LIN {X 0,Y 9.05,Z 814.332,A -85,B 0,C 180,E1 1253.904,E2 1253.904} C_VEL
LIN {X 0,Y 5.338,Z 813.889,A -85,B 0,C 180,E1 1100.52,E2 1100.52} C_VEL
LIN {X 0,Y 12.106,Z 813.495,A -85,B 0,C 180,E1 1087.642,E2 1087.642} C_VEL
LIN {X 0,Y 1.103,Z 814.387,A -85,B 0,C 180,E1 989.979,E2 989.979} C_VEL
LIN {X 0,Y 2.332,Z 814.384,A -85,B 0,C 180,E1 916.768,E2 916.768} C_VEL
LIN {X 0,Y 4.204,Z 816.384,A -85,B 0,C 180,E1 903.517,E2 903.517} C_VEL
LIN {X 0,Y 4.204,Z 862.5,A -85,B 0,C 180,E1 903.517,E2 903.517} C_VEL
LIN {X 0,Y 4.204,Z 862.5,A -85,B 0,C 180,E1 903.517,E2 903.517}

QRS_NEXT_CUT()

QRS_NEXT()
QRS_HOME()

END
